// TIA Portal V17 export
// export: Created 2025-07-01T14:25:34.2784289Z, ExportSetting WithDefaults, DisplayName Totally Integrated Automation Portal, DisplayVersion V17 Update 8, DisplayName TIA Portal Openness, DisplayVersion V17 Update 8, DisplayName TIA Portal Version Control Interface, DisplayVersion V17, DisplayName SINAMICS Startdrive Advanced, DisplayVersion V17 SP2, DisplayName SINAMICS Startdrive G110M, G120, G120C, G120D, G120P, G115D, DisplayVersion V17 SP2, DisplayName SINAMICS Startdrive G130, G150, S120, S150, SINAMICS MV, S210, DisplayVersion V17 SP2, DisplayName STEP 7 Professional, DisplayVersion V17 Update 8, DisplayName SINUMERIK ONE STEP 7 Toolbox, DisplayVersion V17 Update 12, DisplayName SINUMERIK ONE PLC Basic Program Plus, DisplayVersion V17 Update 12, DisplayName SINUMERIK 840D sl STEP 7 Toolbox, DisplayVersion V17 Update 12, DisplayName STEP 7 Safety, DisplayVersion V17 Update 6, DisplayName WinCC Advanced, DisplayVersion V17 Update 8
FUNCTION "FC343_NCK_M_CH1_UNIT_1_STA_0" : Void   // FC343, LAD
TITLE = Channel 1 data
{ S7_Optimized_Access := 'FALSE' }
AUTHOR : ETXETAR
VERSION : 1.0
// stored: AutoNumber false, IsIECCheckEnabled false, SetENOAutomatically false, UDAEnableTagReadback false
BEGIN

REGION Network 1: ACKNOWLEDGE M704-UNIT 1 FIXTURE 4 VERIFY PART AND TOOL IS CLAMPED DURING MACHINING (WHEN TRUE DO). TOGGLED / ACKNOWLEDGE M46-VERIFY FIXTURE 1 PART AND TOOL IS CLAMPED DURING
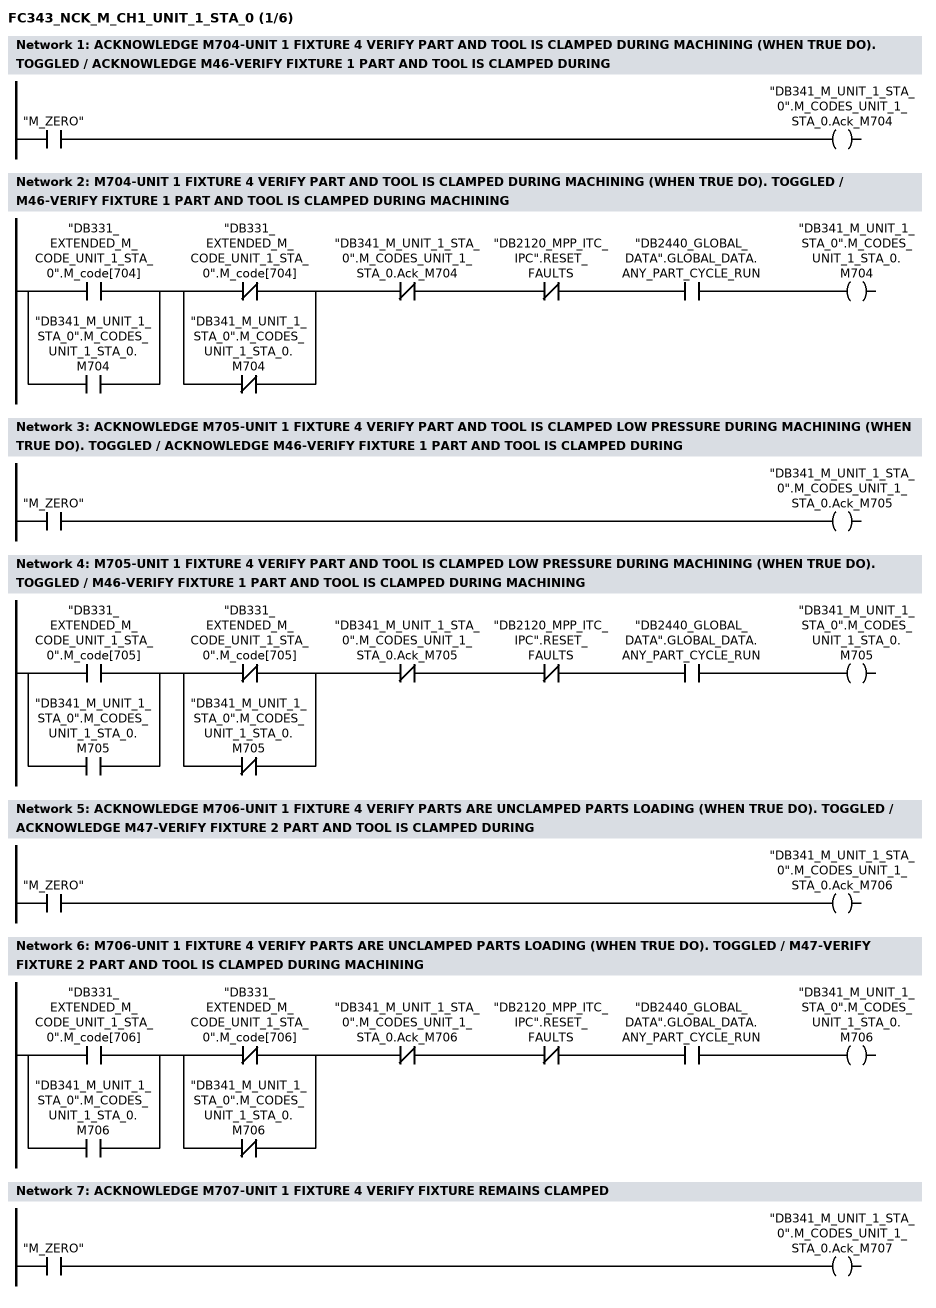
   RUNG wire#powerrail
      Contact( "M_ZERO" )
      Coil( "DB341_M_UNIT_1_STA_0".M_CODES_UNIT_1_STA_0.Ack_M704 )
   END_RUNG
   // the same network as SCL:
   "DB341_M_UNIT_1_STA_0".M_CODES_UNIT_1_STA_0.Ack_M704 := "M_ZERO";
END_REGION

REGION Network 2: M704-UNIT 1 FIXTURE 4 VERIFY PART AND TOOL IS CLAMPED DURING MACHINING (WHEN TRUE DO). TOGGLED / M46-VERIFY FIXTURE 1 PART AND TOOL IS CLAMPED DURING MACHINING
   RUNG wire#powerrail
      Contact( "DB331_EXTENDED_M_CODE_UNIT_1_STA_0".M_code[704] )
      wire#w1
      I_Contact( "DB331_EXTENDED_M_CODE_UNIT_1_STA_0".M_code[704] )
      wire#w2
      I_Contact( "DB341_M_UNIT_1_STA_0".M_CODES_UNIT_1_STA_0.Ack_M704 )
      I_Contact( "DB2120_MPP_ITC_IPC".RESET_FAULTS )
      Contact( "DB2440_GLOBAL_DATA".GLOBAL_DATA.ANY_PART_CYCLE_RUN )
      Coil( "DB341_M_UNIT_1_STA_0".M_CODES_UNIT_1_STA_0.M704 )
   END_RUNG
   RUNG wire#powerrail
      Contact( "DB341_M_UNIT_1_STA_0".M_CODES_UNIT_1_STA_0.M704 )
   END_RUNG wire#w1
   RUNG wire#w1
      I_Contact( "DB341_M_UNIT_1_STA_0".M_CODES_UNIT_1_STA_0.M704 )
   END_RUNG wire#w2
   // the same network as SCL:
   "DB341_M_UNIT_1_STA_0".M_CODES_UNIT_1_STA_0.M704 := ("DB331_EXTENDED_M_CODE_UNIT_1_STA_0".M_code[704] OR "DB341_M_UNIT_1_STA_0".M_CODES_UNIT_1_STA_0.M704) AND (NOT "DB331_EXTENDED_M_CODE_UNIT_1_STA_0".M_code[704] OR NOT "DB341_M_UNIT_1_STA_0".M_CODES_UNIT_1_STA_0.M704) AND NOT "DB341_M_UNIT_1_STA_0".M_CODES_UNIT_1_STA_0.Ack_M704 AND NOT "DB2120_MPP_ITC_IPC".RESET_FAULTS AND "DB2440_GLOBAL_DATA".GLOBAL_DATA.ANY_PART_CYCLE_RUN;
END_REGION

REGION Network 3: ACKNOWLEDGE M705-UNIT 1 FIXTURE 4 VERIFY PART AND TOOL IS CLAMPED LOW PRESSURE DURING MACHINING (WHEN TRUE DO). TOGGLED / ACKNOWLEDGE M46-VERIFY FIXTURE 1 PART AND TOOL IS CLAMPED DURING
   RUNG wire#powerrail
      Contact( "M_ZERO" )
      Coil( "DB341_M_UNIT_1_STA_0".M_CODES_UNIT_1_STA_0.Ack_M705 )
   END_RUNG
   // the same network as SCL:
   "DB341_M_UNIT_1_STA_0".M_CODES_UNIT_1_STA_0.Ack_M705 := "M_ZERO";
END_REGION

REGION Network 4: M705-UNIT 1 FIXTURE 4 VERIFY PART AND TOOL IS CLAMPED LOW PRESSURE DURING MACHINING (WHEN TRUE DO). TOGGLED / M46-VERIFY FIXTURE 1 PART AND TOOL IS CLAMPED DURING MACHINING
   RUNG wire#powerrail
      Contact( "DB331_EXTENDED_M_CODE_UNIT_1_STA_0".M_code[705] )
      wire#w1
      I_Contact( "DB331_EXTENDED_M_CODE_UNIT_1_STA_0".M_code[705] )
      wire#w2
      I_Contact( "DB341_M_UNIT_1_STA_0".M_CODES_UNIT_1_STA_0.Ack_M705 )
      I_Contact( "DB2120_MPP_ITC_IPC".RESET_FAULTS )
      Contact( "DB2440_GLOBAL_DATA".GLOBAL_DATA.ANY_PART_CYCLE_RUN )
      Coil( "DB341_M_UNIT_1_STA_0".M_CODES_UNIT_1_STA_0.M705 )
   END_RUNG
   RUNG wire#powerrail
      Contact( "DB341_M_UNIT_1_STA_0".M_CODES_UNIT_1_STA_0.M705 )
   END_RUNG wire#w1
   RUNG wire#w1
      I_Contact( "DB341_M_UNIT_1_STA_0".M_CODES_UNIT_1_STA_0.M705 )
   END_RUNG wire#w2
   // the same network as SCL:
   "DB341_M_UNIT_1_STA_0".M_CODES_UNIT_1_STA_0.M705 := ("DB331_EXTENDED_M_CODE_UNIT_1_STA_0".M_code[705] OR "DB341_M_UNIT_1_STA_0".M_CODES_UNIT_1_STA_0.M705) AND (NOT "DB331_EXTENDED_M_CODE_UNIT_1_STA_0".M_code[705] OR NOT "DB341_M_UNIT_1_STA_0".M_CODES_UNIT_1_STA_0.M705) AND NOT "DB341_M_UNIT_1_STA_0".M_CODES_UNIT_1_STA_0.Ack_M705 AND NOT "DB2120_MPP_ITC_IPC".RESET_FAULTS AND "DB2440_GLOBAL_DATA".GLOBAL_DATA.ANY_PART_CYCLE_RUN;
END_REGION

REGION Network 5: ACKNOWLEDGE M706-UNIT 1 FIXTURE 4 VERIFY PARTS ARE UNCLAMPED PARTS LOADING (WHEN TRUE DO). TOGGLED / ACKNOWLEDGE M47-VERIFY FIXTURE 2 PART AND TOOL IS CLAMPED DURING
   RUNG wire#powerrail
      Contact( "M_ZERO" )
      Coil( "DB341_M_UNIT_1_STA_0".M_CODES_UNIT_1_STA_0.Ack_M706 )
   END_RUNG
   // the same network as SCL:
   "DB341_M_UNIT_1_STA_0".M_CODES_UNIT_1_STA_0.Ack_M706 := "M_ZERO";
END_REGION

REGION Network 6: M706-UNIT 1 FIXTURE 4 VERIFY PARTS ARE UNCLAMPED PARTS LOADING (WHEN TRUE DO). TOGGLED / M47-VERIFY FIXTURE 2 PART AND TOOL IS CLAMPED DURING MACHINING
   RUNG wire#powerrail
      Contact( "DB331_EXTENDED_M_CODE_UNIT_1_STA_0".M_code[706] )
      wire#w1
      I_Contact( "DB331_EXTENDED_M_CODE_UNIT_1_STA_0".M_code[706] )
      wire#w2
      I_Contact( "DB341_M_UNIT_1_STA_0".M_CODES_UNIT_1_STA_0.Ack_M706 )
      I_Contact( "DB2120_MPP_ITC_IPC".RESET_FAULTS )
      Contact( "DB2440_GLOBAL_DATA".GLOBAL_DATA.ANY_PART_CYCLE_RUN )
      Coil( "DB341_M_UNIT_1_STA_0".M_CODES_UNIT_1_STA_0.M706 )
   END_RUNG
   RUNG wire#powerrail
      Contact( "DB341_M_UNIT_1_STA_0".M_CODES_UNIT_1_STA_0.M706 )
   END_RUNG wire#w1
   RUNG wire#w1
      I_Contact( "DB341_M_UNIT_1_STA_0".M_CODES_UNIT_1_STA_0.M706 )
   END_RUNG wire#w2
   // the same network as SCL:
   "DB341_M_UNIT_1_STA_0".M_CODES_UNIT_1_STA_0.M706 := ("DB331_EXTENDED_M_CODE_UNIT_1_STA_0".M_code[706] OR "DB341_M_UNIT_1_STA_0".M_CODES_UNIT_1_STA_0.M706) AND (NOT "DB331_EXTENDED_M_CODE_UNIT_1_STA_0".M_code[706] OR NOT "DB341_M_UNIT_1_STA_0".M_CODES_UNIT_1_STA_0.M706) AND NOT "DB341_M_UNIT_1_STA_0".M_CODES_UNIT_1_STA_0.Ack_M706 AND NOT "DB2120_MPP_ITC_IPC".RESET_FAULTS AND "DB2440_GLOBAL_DATA".GLOBAL_DATA.ANY_PART_CYCLE_RUN;
END_REGION

REGION Network 7: ACKNOWLEDGE M707-UNIT 1 FIXTURE 4 VERIFY FIXTURE REMAINS CLAMPED
   RUNG wire#powerrail
      Contact( "M_ZERO" )
      Coil( "DB341_M_UNIT_1_STA_0".M_CODES_UNIT_1_STA_0.Ack_M707 )
   END_RUNG
   // the same network as SCL:
   "DB341_M_UNIT_1_STA_0".M_CODES_UNIT_1_STA_0.Ack_M707 := "M_ZERO";
END_REGION

REGION Network 8: M707-UNIT 1 FIXTURE 4 VERIFY FIXTURE REMAINS CLAMPED
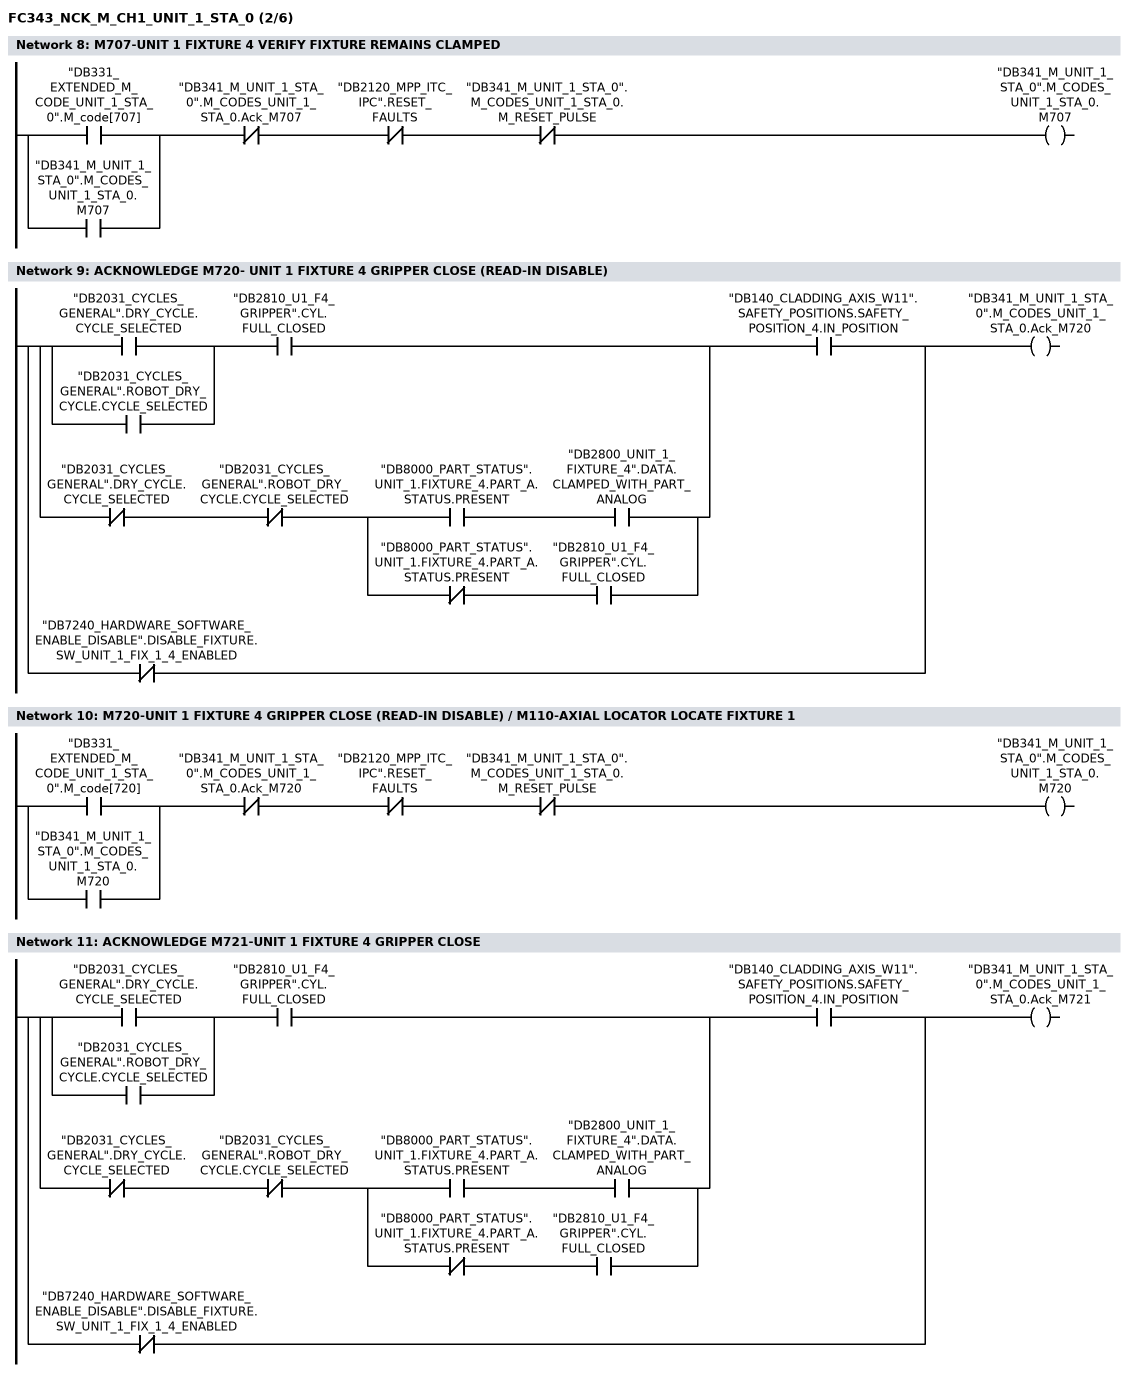
   RUNG wire#powerrail
      Contact( "DB331_EXTENDED_M_CODE_UNIT_1_STA_0".M_code[707] )
      wire#w1
      I_Contact( "DB341_M_UNIT_1_STA_0".M_CODES_UNIT_1_STA_0.Ack_M707 )
      I_Contact( "DB2120_MPP_ITC_IPC".RESET_FAULTS )
      I_Contact( "DB341_M_UNIT_1_STA_0".M_CODES_UNIT_1_STA_0.M_RESET_PULSE )
      Coil( "DB341_M_UNIT_1_STA_0".M_CODES_UNIT_1_STA_0.M707 )
   END_RUNG
   RUNG wire#powerrail
      Contact( "DB341_M_UNIT_1_STA_0".M_CODES_UNIT_1_STA_0.M707 )
   END_RUNG wire#w1
   // the same network as SCL:
   "DB341_M_UNIT_1_STA_0".M_CODES_UNIT_1_STA_0.M707 := ("DB331_EXTENDED_M_CODE_UNIT_1_STA_0".M_code[707] OR "DB341_M_UNIT_1_STA_0".M_CODES_UNIT_1_STA_0.M707) AND NOT "DB341_M_UNIT_1_STA_0".M_CODES_UNIT_1_STA_0.Ack_M707 AND NOT "DB2120_MPP_ITC_IPC".RESET_FAULTS AND NOT "DB341_M_UNIT_1_STA_0".M_CODES_UNIT_1_STA_0.M_RESET_PULSE;
END_REGION

REGION Network 9: ACKNOWLEDGE M720- UNIT 1 FIXTURE 4 GRIPPER CLOSE (READ-IN DISABLE)
   RUNG wire#powerrail
      Contact( "DB2031_CYCLES_GENERAL".DRY_CYCLE.CYCLE_SELECTED )
      wire#w1
      Contact( "DB2810_U1_F4_GRIPPER".CYL.FULL_CLOSED )
      wire#w2
      Contact( "DB140_CLADDING_AXIS_W11".SAFETY_POSITIONS.SAFETY_POSITION_4.IN_POSITION )
      wire#w4
      Coil( "DB341_M_UNIT_1_STA_0".M_CODES_UNIT_1_STA_0.Ack_M720 )
   END_RUNG
   RUNG wire#powerrail
      Contact( "DB2031_CYCLES_GENERAL".ROBOT_DRY_CYCLE.CYCLE_SELECTED )
   END_RUNG wire#w1
   RUNG wire#powerrail
      I_Contact( "DB2031_CYCLES_GENERAL".DRY_CYCLE.CYCLE_SELECTED )
      I_Contact( "DB2031_CYCLES_GENERAL".ROBOT_DRY_CYCLE.CYCLE_SELECTED )
      wire#w3
      Contact( "DB8000_PART_STATUS".UNIT_1.FIXTURE_4.PART_A.STATUS.PRESENT )
      Contact( "DB2800_UNIT_1_FIXTURE_4".DATA.CLAMPED_WITH_PART_ANALOG )
   END_RUNG wire#w2
   RUNG wire#w3
      I_Contact( "DB8000_PART_STATUS".UNIT_1.FIXTURE_4.PART_A.STATUS.PRESENT )
      Contact( "DB2810_U1_F4_GRIPPER".CYL.FULL_CLOSED )
   END_RUNG wire#w2
   RUNG wire#powerrail
      I_Contact( "DB7240_HARDWARE_SOFTWARE_ENABLE_DISABLE".DISABLE_FIXTURE.SW_UNIT_1_FIX_1_4_ENABLED )
   END_RUNG wire#w4
   // the same network as SCL:
   "DB341_M_UNIT_1_STA_0".M_CODES_UNIT_1_STA_0.Ack_M720 := (((("DB2031_CYCLES_GENERAL".DRY_CYCLE.CYCLE_SELECTED OR "DB2031_CYCLES_GENERAL".ROBOT_DRY_CYCLE.CYCLE_SELECTED) AND "DB2810_U1_F4_GRIPPER".CYL.FULL_CLOSED) OR (NOT "DB2031_CYCLES_GENERAL".DRY_CYCLE.CYCLE_SELECTED AND NOT "DB2031_CYCLES_GENERAL".ROBOT_DRY_CYCLE.CYCLE_SELECTED AND (("DB8000_PART_STATUS".UNIT_1.FIXTURE_4.PART_A.STATUS.PRESENT AND "DB2800_UNIT_1_FIXTURE_4".DATA.CLAMPED_WITH_PART_ANALOG) OR (NOT "DB8000_PART_STATUS".UNIT_1.FIXTURE_4.PART_A.STATUS.PRESENT AND "DB2810_U1_F4_GRIPPER".CYL.FULL_CLOSED)))) AND "DB140_CLADDING_AXIS_W11".SAFETY_POSITIONS.SAFETY_POSITION_4.IN_POSITION) OR NOT "DB7240_HARDWARE_SOFTWARE_ENABLE_DISABLE".DISABLE_FIXTURE.SW_UNIT_1_FIX_1_4_ENABLED;
END_REGION

REGION Network 10: M720-UNIT 1 FIXTURE 4 GRIPPER CLOSE (READ-IN DISABLE) / M110-AXIAL LOCATOR LOCATE FIXTURE 1
   RUNG wire#powerrail
      Contact( "DB331_EXTENDED_M_CODE_UNIT_1_STA_0".M_code[720] )
      wire#w1
      I_Contact( "DB341_M_UNIT_1_STA_0".M_CODES_UNIT_1_STA_0.Ack_M720 )
      I_Contact( "DB2120_MPP_ITC_IPC".RESET_FAULTS )
      I_Contact( "DB341_M_UNIT_1_STA_0".M_CODES_UNIT_1_STA_0.M_RESET_PULSE )
      Coil( "DB341_M_UNIT_1_STA_0".M_CODES_UNIT_1_STA_0.M720 )
   END_RUNG
   RUNG wire#powerrail
      Contact( "DB341_M_UNIT_1_STA_0".M_CODES_UNIT_1_STA_0.M720 )
   END_RUNG wire#w1
   // the same network as SCL:
   "DB341_M_UNIT_1_STA_0".M_CODES_UNIT_1_STA_0.M720 := ("DB331_EXTENDED_M_CODE_UNIT_1_STA_0".M_code[720] OR "DB341_M_UNIT_1_STA_0".M_CODES_UNIT_1_STA_0.M720) AND NOT "DB341_M_UNIT_1_STA_0".M_CODES_UNIT_1_STA_0.Ack_M720 AND NOT "DB2120_MPP_ITC_IPC".RESET_FAULTS AND NOT "DB341_M_UNIT_1_STA_0".M_CODES_UNIT_1_STA_0.M_RESET_PULSE;
END_REGION

REGION Network 11: ACKNOWLEDGE M721-UNIT 1 FIXTURE 4 GRIPPER CLOSE
   RUNG wire#powerrail
      Contact( "DB2031_CYCLES_GENERAL".DRY_CYCLE.CYCLE_SELECTED )
      wire#w1
      Contact( "DB2810_U1_F4_GRIPPER".CYL.FULL_CLOSED )
      wire#w2
      Contact( "DB140_CLADDING_AXIS_W11".SAFETY_POSITIONS.SAFETY_POSITION_4.IN_POSITION )
      wire#w4
      Coil( "DB341_M_UNIT_1_STA_0".M_CODES_UNIT_1_STA_0.Ack_M721 )
   END_RUNG
   RUNG wire#powerrail
      Contact( "DB2031_CYCLES_GENERAL".ROBOT_DRY_CYCLE.CYCLE_SELECTED )
   END_RUNG wire#w1
   RUNG wire#powerrail
      I_Contact( "DB2031_CYCLES_GENERAL".DRY_CYCLE.CYCLE_SELECTED )
      I_Contact( "DB2031_CYCLES_GENERAL".ROBOT_DRY_CYCLE.CYCLE_SELECTED )
      wire#w3
      Contact( "DB8000_PART_STATUS".UNIT_1.FIXTURE_4.PART_A.STATUS.PRESENT )
      Contact( "DB2800_UNIT_1_FIXTURE_4".DATA.CLAMPED_WITH_PART_ANALOG )
   END_RUNG wire#w2
   RUNG wire#w3
      I_Contact( "DB8000_PART_STATUS".UNIT_1.FIXTURE_4.PART_A.STATUS.PRESENT )
      Contact( "DB2810_U1_F4_GRIPPER".CYL.FULL_CLOSED )
   END_RUNG wire#w2
   RUNG wire#powerrail
      I_Contact( "DB7240_HARDWARE_SOFTWARE_ENABLE_DISABLE".DISABLE_FIXTURE.SW_UNIT_1_FIX_1_4_ENABLED )
   END_RUNG wire#w4
   // the same network as SCL:
   "DB341_M_UNIT_1_STA_0".M_CODES_UNIT_1_STA_0.Ack_M721 := (((("DB2031_CYCLES_GENERAL".DRY_CYCLE.CYCLE_SELECTED OR "DB2031_CYCLES_GENERAL".ROBOT_DRY_CYCLE.CYCLE_SELECTED) AND "DB2810_U1_F4_GRIPPER".CYL.FULL_CLOSED) OR (NOT "DB2031_CYCLES_GENERAL".DRY_CYCLE.CYCLE_SELECTED AND NOT "DB2031_CYCLES_GENERAL".ROBOT_DRY_CYCLE.CYCLE_SELECTED AND (("DB8000_PART_STATUS".UNIT_1.FIXTURE_4.PART_A.STATUS.PRESENT AND "DB2800_UNIT_1_FIXTURE_4".DATA.CLAMPED_WITH_PART_ANALOG) OR (NOT "DB8000_PART_STATUS".UNIT_1.FIXTURE_4.PART_A.STATUS.PRESENT AND "DB2810_U1_F4_GRIPPER".CYL.FULL_CLOSED)))) AND "DB140_CLADDING_AXIS_W11".SAFETY_POSITIONS.SAFETY_POSITION_4.IN_POSITION) OR NOT "DB7240_HARDWARE_SOFTWARE_ENABLE_DISABLE".DISABLE_FIXTURE.SW_UNIT_1_FIX_1_4_ENABLED;
END_REGION

REGION Network 12: M721-UNIT 1 FIXTURE 4 GRIPPER CLOSE / M110-AXIAL LOCATOR LOCATE FIXTURE 1
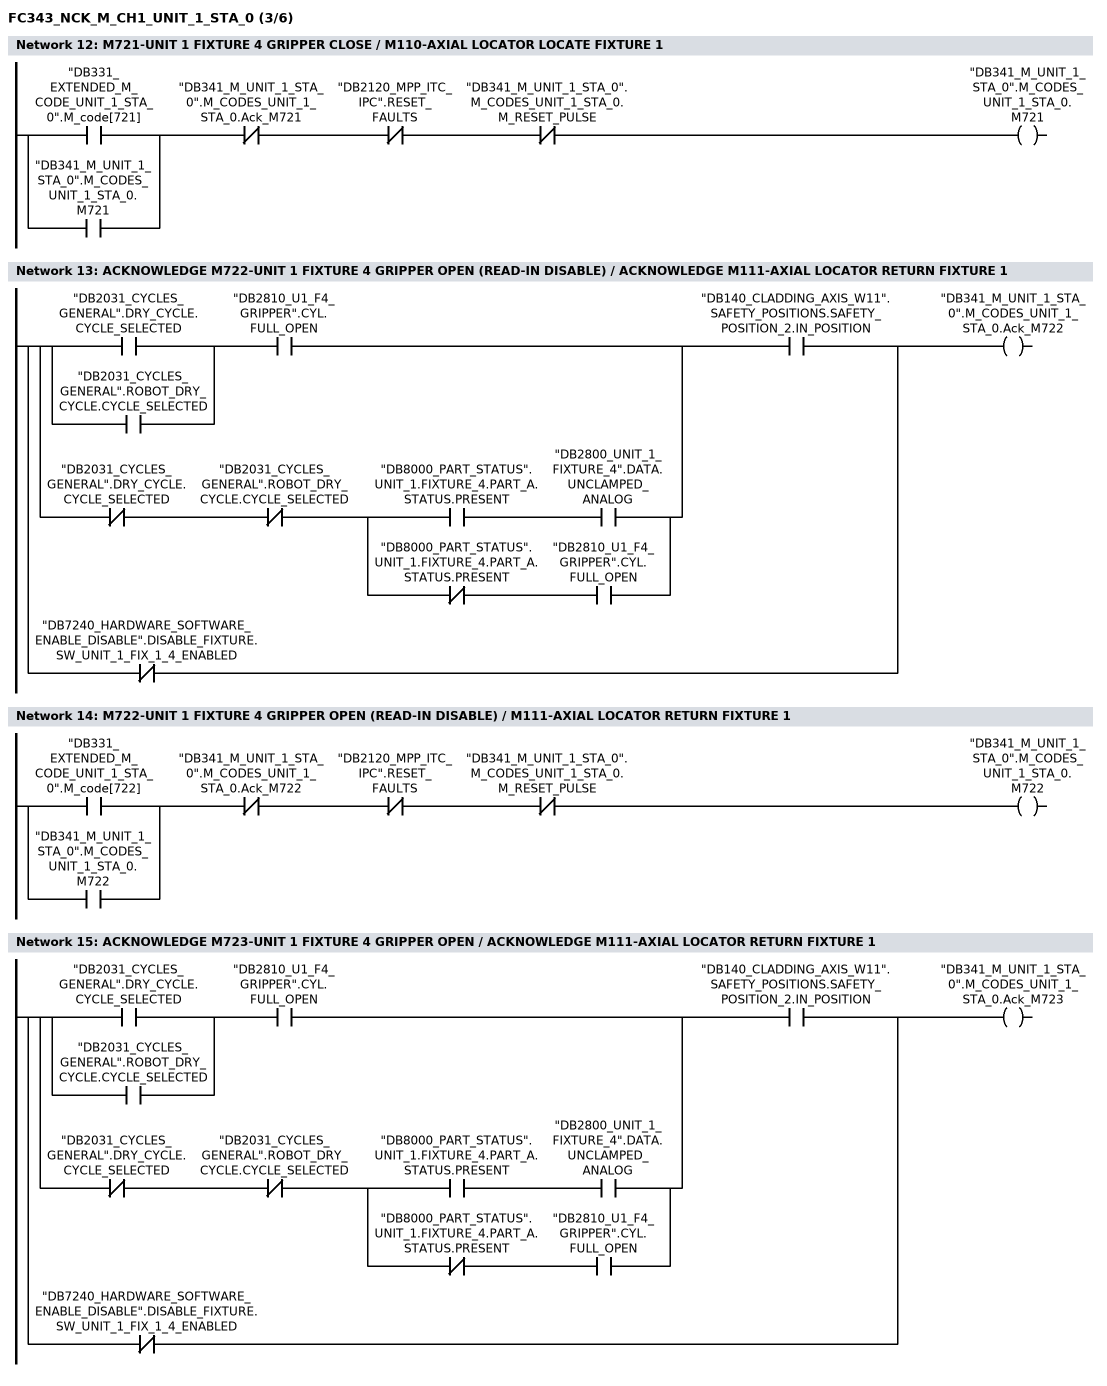
   RUNG wire#powerrail
      Contact( "DB331_EXTENDED_M_CODE_UNIT_1_STA_0".M_code[721] )
      wire#w1
      I_Contact( "DB341_M_UNIT_1_STA_0".M_CODES_UNIT_1_STA_0.Ack_M721 )
      I_Contact( "DB2120_MPP_ITC_IPC".RESET_FAULTS )
      I_Contact( "DB341_M_UNIT_1_STA_0".M_CODES_UNIT_1_STA_0.M_RESET_PULSE )
      Coil( "DB341_M_UNIT_1_STA_0".M_CODES_UNIT_1_STA_0.M721 )
   END_RUNG
   RUNG wire#powerrail
      Contact( "DB341_M_UNIT_1_STA_0".M_CODES_UNIT_1_STA_0.M721 )
   END_RUNG wire#w1
   // the same network as SCL:
   "DB341_M_UNIT_1_STA_0".M_CODES_UNIT_1_STA_0.M721 := ("DB331_EXTENDED_M_CODE_UNIT_1_STA_0".M_code[721] OR "DB341_M_UNIT_1_STA_0".M_CODES_UNIT_1_STA_0.M721) AND NOT "DB341_M_UNIT_1_STA_0".M_CODES_UNIT_1_STA_0.Ack_M721 AND NOT "DB2120_MPP_ITC_IPC".RESET_FAULTS AND NOT "DB341_M_UNIT_1_STA_0".M_CODES_UNIT_1_STA_0.M_RESET_PULSE;
END_REGION

REGION Network 13: ACKNOWLEDGE M722-UNIT 1 FIXTURE 4 GRIPPER OPEN (READ-IN DISABLE) / ACKNOWLEDGE M111-AXIAL LOCATOR RETURN FIXTURE 1
   RUNG wire#powerrail
      Contact( "DB2031_CYCLES_GENERAL".DRY_CYCLE.CYCLE_SELECTED )
      wire#w1
      Contact( "DB2810_U1_F4_GRIPPER".CYL.FULL_OPEN )
      wire#w2
      Contact( "DB140_CLADDING_AXIS_W11".SAFETY_POSITIONS.SAFETY_POSITION_2.IN_POSITION )
      wire#w4
      Coil( "DB341_M_UNIT_1_STA_0".M_CODES_UNIT_1_STA_0.Ack_M722 )
   END_RUNG
   RUNG wire#powerrail
      Contact( "DB2031_CYCLES_GENERAL".ROBOT_DRY_CYCLE.CYCLE_SELECTED )
   END_RUNG wire#w1
   RUNG wire#powerrail
      I_Contact( "DB2031_CYCLES_GENERAL".DRY_CYCLE.CYCLE_SELECTED )
      I_Contact( "DB2031_CYCLES_GENERAL".ROBOT_DRY_CYCLE.CYCLE_SELECTED )
      wire#w3
      Contact( "DB8000_PART_STATUS".UNIT_1.FIXTURE_4.PART_A.STATUS.PRESENT )
      Contact( "DB2800_UNIT_1_FIXTURE_4".DATA.UNCLAMPED_ANALOG )
   END_RUNG wire#w2
   RUNG wire#w3
      I_Contact( "DB8000_PART_STATUS".UNIT_1.FIXTURE_4.PART_A.STATUS.PRESENT )
      Contact( "DB2810_U1_F4_GRIPPER".CYL.FULL_OPEN )
   END_RUNG wire#w2
   RUNG wire#powerrail
      I_Contact( "DB7240_HARDWARE_SOFTWARE_ENABLE_DISABLE".DISABLE_FIXTURE.SW_UNIT_1_FIX_1_4_ENABLED )
   END_RUNG wire#w4
   // the same network as SCL:
   "DB341_M_UNIT_1_STA_0".M_CODES_UNIT_1_STA_0.Ack_M722 := (((("DB2031_CYCLES_GENERAL".DRY_CYCLE.CYCLE_SELECTED OR "DB2031_CYCLES_GENERAL".ROBOT_DRY_CYCLE.CYCLE_SELECTED) AND "DB2810_U1_F4_GRIPPER".CYL.FULL_OPEN) OR (NOT "DB2031_CYCLES_GENERAL".DRY_CYCLE.CYCLE_SELECTED AND NOT "DB2031_CYCLES_GENERAL".ROBOT_DRY_CYCLE.CYCLE_SELECTED AND (("DB8000_PART_STATUS".UNIT_1.FIXTURE_4.PART_A.STATUS.PRESENT AND "DB2800_UNIT_1_FIXTURE_4".DATA.UNCLAMPED_ANALOG) OR (NOT "DB8000_PART_STATUS".UNIT_1.FIXTURE_4.PART_A.STATUS.PRESENT AND "DB2810_U1_F4_GRIPPER".CYL.FULL_OPEN)))) AND "DB140_CLADDING_AXIS_W11".SAFETY_POSITIONS.SAFETY_POSITION_2.IN_POSITION) OR NOT "DB7240_HARDWARE_SOFTWARE_ENABLE_DISABLE".DISABLE_FIXTURE.SW_UNIT_1_FIX_1_4_ENABLED;
END_REGION

REGION Network 14: M722-UNIT 1 FIXTURE 4 GRIPPER OPEN (READ-IN DISABLE) / M111-AXIAL LOCATOR RETURN FIXTURE 1
   RUNG wire#powerrail
      Contact( "DB331_EXTENDED_M_CODE_UNIT_1_STA_0".M_code[722] )
      wire#w1
      I_Contact( "DB341_M_UNIT_1_STA_0".M_CODES_UNIT_1_STA_0.Ack_M722 )
      I_Contact( "DB2120_MPP_ITC_IPC".RESET_FAULTS )
      I_Contact( "DB341_M_UNIT_1_STA_0".M_CODES_UNIT_1_STA_0.M_RESET_PULSE )
      Coil( "DB341_M_UNIT_1_STA_0".M_CODES_UNIT_1_STA_0.M722 )
   END_RUNG
   RUNG wire#powerrail
      Contact( "DB341_M_UNIT_1_STA_0".M_CODES_UNIT_1_STA_0.M722 )
   END_RUNG wire#w1
   // the same network as SCL:
   "DB341_M_UNIT_1_STA_0".M_CODES_UNIT_1_STA_0.M722 := ("DB331_EXTENDED_M_CODE_UNIT_1_STA_0".M_code[722] OR "DB341_M_UNIT_1_STA_0".M_CODES_UNIT_1_STA_0.M722) AND NOT "DB341_M_UNIT_1_STA_0".M_CODES_UNIT_1_STA_0.Ack_M722 AND NOT "DB2120_MPP_ITC_IPC".RESET_FAULTS AND NOT "DB341_M_UNIT_1_STA_0".M_CODES_UNIT_1_STA_0.M_RESET_PULSE;
END_REGION

REGION Network 15: ACKNOWLEDGE M723-UNIT 1 FIXTURE 4 GRIPPER OPEN / ACKNOWLEDGE M111-AXIAL LOCATOR RETURN FIXTURE 1
   RUNG wire#powerrail
      Contact( "DB2031_CYCLES_GENERAL".DRY_CYCLE.CYCLE_SELECTED )
      wire#w1
      Contact( "DB2810_U1_F4_GRIPPER".CYL.FULL_OPEN )
      wire#w2
      Contact( "DB140_CLADDING_AXIS_W11".SAFETY_POSITIONS.SAFETY_POSITION_2.IN_POSITION )
      wire#w4
      Coil( "DB341_M_UNIT_1_STA_0".M_CODES_UNIT_1_STA_0.Ack_M723 )
   END_RUNG
   RUNG wire#powerrail
      Contact( "DB2031_CYCLES_GENERAL".ROBOT_DRY_CYCLE.CYCLE_SELECTED )
   END_RUNG wire#w1
   RUNG wire#powerrail
      I_Contact( "DB2031_CYCLES_GENERAL".DRY_CYCLE.CYCLE_SELECTED )
      I_Contact( "DB2031_CYCLES_GENERAL".ROBOT_DRY_CYCLE.CYCLE_SELECTED )
      wire#w3
      Contact( "DB8000_PART_STATUS".UNIT_1.FIXTURE_4.PART_A.STATUS.PRESENT )
      Contact( "DB2800_UNIT_1_FIXTURE_4".DATA.UNCLAMPED_ANALOG )
   END_RUNG wire#w2
   RUNG wire#w3
      I_Contact( "DB8000_PART_STATUS".UNIT_1.FIXTURE_4.PART_A.STATUS.PRESENT )
      Contact( "DB2810_U1_F4_GRIPPER".CYL.FULL_OPEN )
   END_RUNG wire#w2
   RUNG wire#powerrail
      I_Contact( "DB7240_HARDWARE_SOFTWARE_ENABLE_DISABLE".DISABLE_FIXTURE.SW_UNIT_1_FIX_1_4_ENABLED )
   END_RUNG wire#w4
   // the same network as SCL:
   "DB341_M_UNIT_1_STA_0".M_CODES_UNIT_1_STA_0.Ack_M723 := (((("DB2031_CYCLES_GENERAL".DRY_CYCLE.CYCLE_SELECTED OR "DB2031_CYCLES_GENERAL".ROBOT_DRY_CYCLE.CYCLE_SELECTED) AND "DB2810_U1_F4_GRIPPER".CYL.FULL_OPEN) OR (NOT "DB2031_CYCLES_GENERAL".DRY_CYCLE.CYCLE_SELECTED AND NOT "DB2031_CYCLES_GENERAL".ROBOT_DRY_CYCLE.CYCLE_SELECTED AND (("DB8000_PART_STATUS".UNIT_1.FIXTURE_4.PART_A.STATUS.PRESENT AND "DB2800_UNIT_1_FIXTURE_4".DATA.UNCLAMPED_ANALOG) OR (NOT "DB8000_PART_STATUS".UNIT_1.FIXTURE_4.PART_A.STATUS.PRESENT AND "DB2810_U1_F4_GRIPPER".CYL.FULL_OPEN)))) AND "DB140_CLADDING_AXIS_W11".SAFETY_POSITIONS.SAFETY_POSITION_2.IN_POSITION) OR NOT "DB7240_HARDWARE_SOFTWARE_ENABLE_DISABLE".DISABLE_FIXTURE.SW_UNIT_1_FIX_1_4_ENABLED;
END_REGION

REGION Network 16: M723-UNIT 1 FIXTURE 4 GRIPPER OPEN / M111-AXIAL LOCATOR RETURN FIXTURE 1
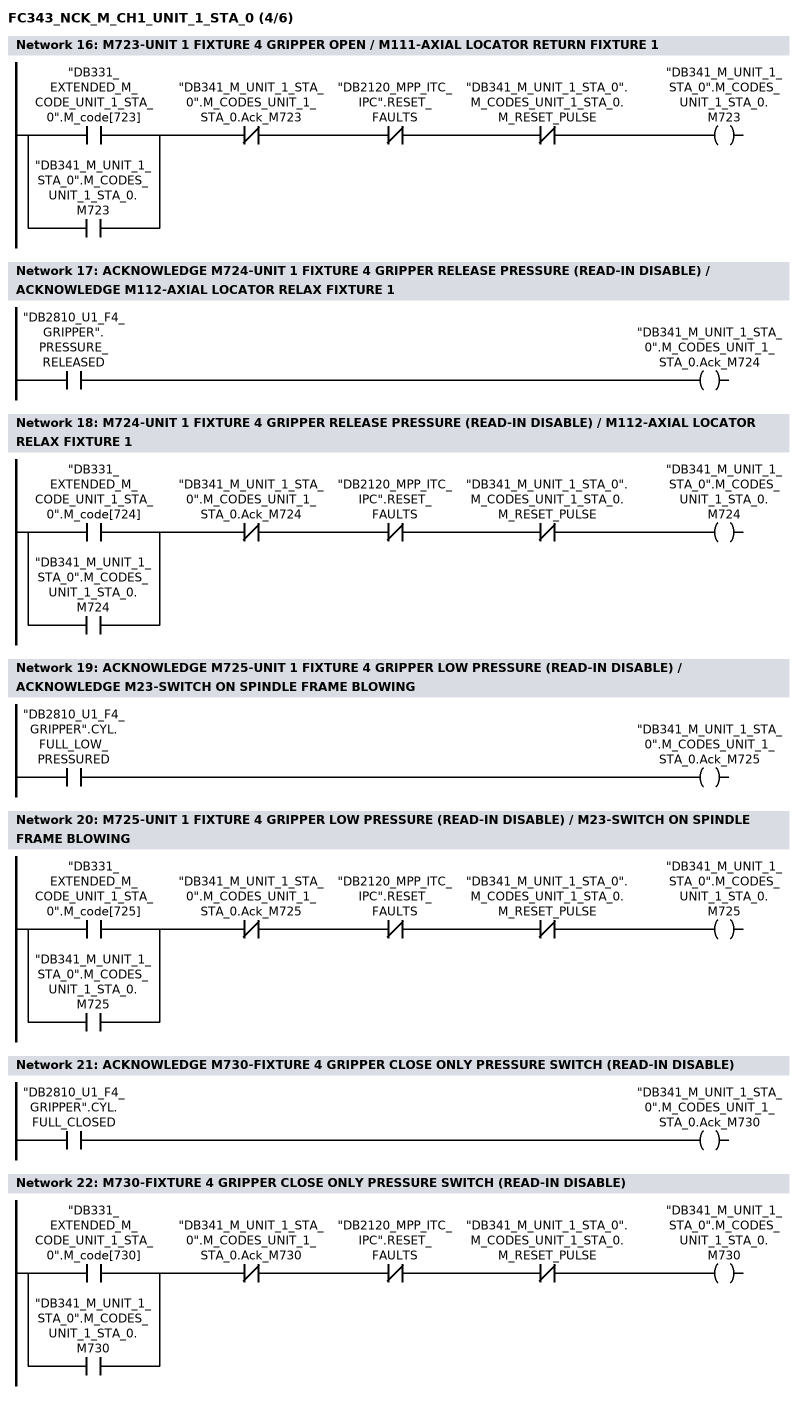
   RUNG wire#powerrail
      Contact( "DB331_EXTENDED_M_CODE_UNIT_1_STA_0".M_code[723] )
      wire#w1
      I_Contact( "DB341_M_UNIT_1_STA_0".M_CODES_UNIT_1_STA_0.Ack_M723 )
      I_Contact( "DB2120_MPP_ITC_IPC".RESET_FAULTS )
      I_Contact( "DB341_M_UNIT_1_STA_0".M_CODES_UNIT_1_STA_0.M_RESET_PULSE )
      Coil( "DB341_M_UNIT_1_STA_0".M_CODES_UNIT_1_STA_0.M723 )
   END_RUNG
   RUNG wire#powerrail
      Contact( "DB341_M_UNIT_1_STA_0".M_CODES_UNIT_1_STA_0.M723 )
   END_RUNG wire#w1
   // the same network as SCL:
   "DB341_M_UNIT_1_STA_0".M_CODES_UNIT_1_STA_0.M723 := ("DB331_EXTENDED_M_CODE_UNIT_1_STA_0".M_code[723] OR "DB341_M_UNIT_1_STA_0".M_CODES_UNIT_1_STA_0.M723) AND NOT "DB341_M_UNIT_1_STA_0".M_CODES_UNIT_1_STA_0.Ack_M723 AND NOT "DB2120_MPP_ITC_IPC".RESET_FAULTS AND NOT "DB341_M_UNIT_1_STA_0".M_CODES_UNIT_1_STA_0.M_RESET_PULSE;
END_REGION

REGION Network 17: ACKNOWLEDGE M724-UNIT 1 FIXTURE 4 GRIPPER RELEASE PRESSURE (READ-IN DISABLE) / ACKNOWLEDGE M112-AXIAL LOCATOR RELAX FIXTURE 1
   RUNG wire#powerrail
      Contact( "DB2810_U1_F4_GRIPPER".PRESSURE_RELEASED )
      Coil( "DB341_M_UNIT_1_STA_0".M_CODES_UNIT_1_STA_0.Ack_M724 )
   END_RUNG
   // the same network as SCL:
   "DB341_M_UNIT_1_STA_0".M_CODES_UNIT_1_STA_0.Ack_M724 := "DB2810_U1_F4_GRIPPER".PRESSURE_RELEASED;
END_REGION

REGION Network 18: M724-UNIT 1 FIXTURE 4 GRIPPER RELEASE PRESSURE (READ-IN DISABLE) / M112-AXIAL LOCATOR RELAX FIXTURE 1
   RUNG wire#powerrail
      Contact( "DB331_EXTENDED_M_CODE_UNIT_1_STA_0".M_code[724] )
      wire#w1
      I_Contact( "DB341_M_UNIT_1_STA_0".M_CODES_UNIT_1_STA_0.Ack_M724 )
      I_Contact( "DB2120_MPP_ITC_IPC".RESET_FAULTS )
      I_Contact( "DB341_M_UNIT_1_STA_0".M_CODES_UNIT_1_STA_0.M_RESET_PULSE )
      Coil( "DB341_M_UNIT_1_STA_0".M_CODES_UNIT_1_STA_0.M724 )
   END_RUNG
   RUNG wire#powerrail
      Contact( "DB341_M_UNIT_1_STA_0".M_CODES_UNIT_1_STA_0.M724 )
   END_RUNG wire#w1
   // the same network as SCL:
   "DB341_M_UNIT_1_STA_0".M_CODES_UNIT_1_STA_0.M724 := ("DB331_EXTENDED_M_CODE_UNIT_1_STA_0".M_code[724] OR "DB341_M_UNIT_1_STA_0".M_CODES_UNIT_1_STA_0.M724) AND NOT "DB341_M_UNIT_1_STA_0".M_CODES_UNIT_1_STA_0.Ack_M724 AND NOT "DB2120_MPP_ITC_IPC".RESET_FAULTS AND NOT "DB341_M_UNIT_1_STA_0".M_CODES_UNIT_1_STA_0.M_RESET_PULSE;
END_REGION

REGION Network 19: ACKNOWLEDGE M725-UNIT 1 FIXTURE 4 GRIPPER LOW PRESSURE (READ-IN DISABLE) / ACKNOWLEDGE M23-SWITCH ON SPINDLE FRAME BLOWING
   RUNG wire#powerrail
      Contact( "DB2810_U1_F4_GRIPPER".CYL.FULL_LOW_PRESSURED )
      Coil( "DB341_M_UNIT_1_STA_0".M_CODES_UNIT_1_STA_0.Ack_M725 )
   END_RUNG
   // the same network as SCL:
   "DB341_M_UNIT_1_STA_0".M_CODES_UNIT_1_STA_0.Ack_M725 := "DB2810_U1_F4_GRIPPER".CYL.FULL_LOW_PRESSURED;
END_REGION

REGION Network 20: M725-UNIT 1 FIXTURE 4 GRIPPER LOW PRESSURE (READ-IN DISABLE) / M23-SWITCH ON SPINDLE FRAME BLOWING
   RUNG wire#powerrail
      Contact( "DB331_EXTENDED_M_CODE_UNIT_1_STA_0".M_code[725] )
      wire#w1
      I_Contact( "DB341_M_UNIT_1_STA_0".M_CODES_UNIT_1_STA_0.Ack_M725 )
      I_Contact( "DB2120_MPP_ITC_IPC".RESET_FAULTS )
      I_Contact( "DB341_M_UNIT_1_STA_0".M_CODES_UNIT_1_STA_0.M_RESET_PULSE )
      Coil( "DB341_M_UNIT_1_STA_0".M_CODES_UNIT_1_STA_0.M725 )
   END_RUNG
   RUNG wire#powerrail
      Contact( "DB341_M_UNIT_1_STA_0".M_CODES_UNIT_1_STA_0.M725 )
   END_RUNG wire#w1
   // the same network as SCL:
   "DB341_M_UNIT_1_STA_0".M_CODES_UNIT_1_STA_0.M725 := ("DB331_EXTENDED_M_CODE_UNIT_1_STA_0".M_code[725] OR "DB341_M_UNIT_1_STA_0".M_CODES_UNIT_1_STA_0.M725) AND NOT "DB341_M_UNIT_1_STA_0".M_CODES_UNIT_1_STA_0.Ack_M725 AND NOT "DB2120_MPP_ITC_IPC".RESET_FAULTS AND NOT "DB341_M_UNIT_1_STA_0".M_CODES_UNIT_1_STA_0.M_RESET_PULSE;
END_REGION

REGION Network 21: ACKNOWLEDGE M730-FIXTURE 4 GRIPPER CLOSE ONLY PRESSURE SWITCH (READ-IN DISABLE)
   RUNG wire#powerrail
      Contact( "DB2810_U1_F4_GRIPPER".CYL.FULL_CLOSED )
      Coil( "DB341_M_UNIT_1_STA_0".M_CODES_UNIT_1_STA_0.Ack_M730 )
   END_RUNG
   // the same network as SCL:
   "DB341_M_UNIT_1_STA_0".M_CODES_UNIT_1_STA_0.Ack_M730 := "DB2810_U1_F4_GRIPPER".CYL.FULL_CLOSED;
END_REGION

REGION Network 22: M730-FIXTURE 4 GRIPPER CLOSE ONLY PRESSURE SWITCH (READ-IN DISABLE)
   RUNG wire#powerrail
      Contact( "DB331_EXTENDED_M_CODE_UNIT_1_STA_0".M_code[730] )
      wire#w1
      I_Contact( "DB341_M_UNIT_1_STA_0".M_CODES_UNIT_1_STA_0.Ack_M730 )
      I_Contact( "DB2120_MPP_ITC_IPC".RESET_FAULTS )
      I_Contact( "DB341_M_UNIT_1_STA_0".M_CODES_UNIT_1_STA_0.M_RESET_PULSE )
      Coil( "DB341_M_UNIT_1_STA_0".M_CODES_UNIT_1_STA_0.M730 )
   END_RUNG
   RUNG wire#powerrail
      Contact( "DB341_M_UNIT_1_STA_0".M_CODES_UNIT_1_STA_0.M730 )
   END_RUNG wire#w1
   // the same network as SCL:
   "DB341_M_UNIT_1_STA_0".M_CODES_UNIT_1_STA_0.M730 := ("DB331_EXTENDED_M_CODE_UNIT_1_STA_0".M_code[730] OR "DB341_M_UNIT_1_STA_0".M_CODES_UNIT_1_STA_0.M730) AND NOT "DB341_M_UNIT_1_STA_0".M_CODES_UNIT_1_STA_0.Ack_M730 AND NOT "DB2120_MPP_ITC_IPC".RESET_FAULTS AND NOT "DB341_M_UNIT_1_STA_0".M_CODES_UNIT_1_STA_0.M_RESET_PULSE;
END_REGION

REGION Network 23: ACKNOWLEDGE M731-FIXTURE 4 GRIPPER CLOSE ONLY PRESSURE SWITCH / ACKNOWLEDGE M23-SWITCH ON SPINDLE FRAME BLOWING
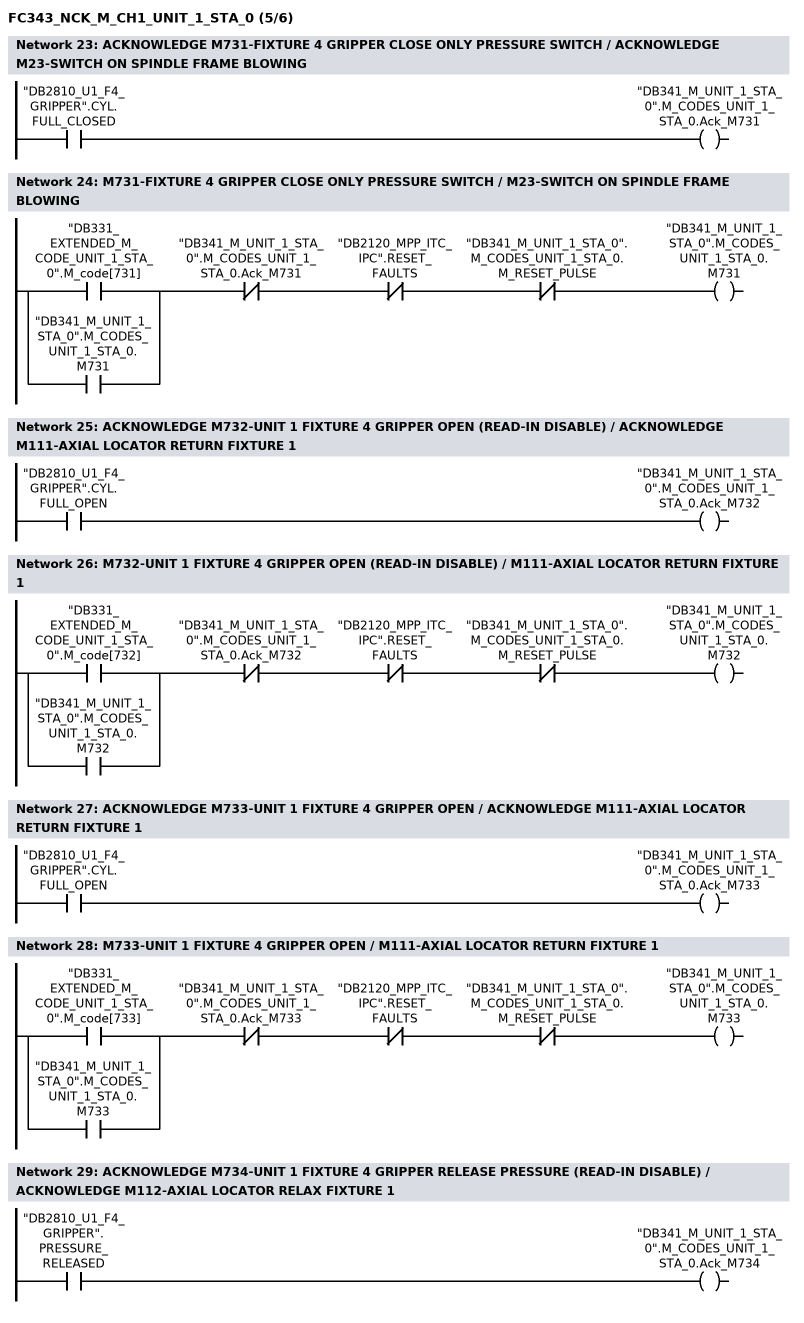
   RUNG wire#powerrail
      Contact( "DB2810_U1_F4_GRIPPER".CYL.FULL_CLOSED )
      Coil( "DB341_M_UNIT_1_STA_0".M_CODES_UNIT_1_STA_0.Ack_M731 )
   END_RUNG
   // the same network as SCL:
   "DB341_M_UNIT_1_STA_0".M_CODES_UNIT_1_STA_0.Ack_M731 := "DB2810_U1_F4_GRIPPER".CYL.FULL_CLOSED;
END_REGION

REGION Network 24: M731-FIXTURE 4 GRIPPER CLOSE ONLY PRESSURE SWITCH / M23-SWITCH ON SPINDLE FRAME BLOWING
   RUNG wire#powerrail
      Contact( "DB331_EXTENDED_M_CODE_UNIT_1_STA_0".M_code[731] )
      wire#w1
      I_Contact( "DB341_M_UNIT_1_STA_0".M_CODES_UNIT_1_STA_0.Ack_M731 )
      I_Contact( "DB2120_MPP_ITC_IPC".RESET_FAULTS )
      I_Contact( "DB341_M_UNIT_1_STA_0".M_CODES_UNIT_1_STA_0.M_RESET_PULSE )
      Coil( "DB341_M_UNIT_1_STA_0".M_CODES_UNIT_1_STA_0.M731 )
   END_RUNG
   RUNG wire#powerrail
      Contact( "DB341_M_UNIT_1_STA_0".M_CODES_UNIT_1_STA_0.M731 )
   END_RUNG wire#w1
   // the same network as SCL:
   "DB341_M_UNIT_1_STA_0".M_CODES_UNIT_1_STA_0.M731 := ("DB331_EXTENDED_M_CODE_UNIT_1_STA_0".M_code[731] OR "DB341_M_UNIT_1_STA_0".M_CODES_UNIT_1_STA_0.M731) AND NOT "DB341_M_UNIT_1_STA_0".M_CODES_UNIT_1_STA_0.Ack_M731 AND NOT "DB2120_MPP_ITC_IPC".RESET_FAULTS AND NOT "DB341_M_UNIT_1_STA_0".M_CODES_UNIT_1_STA_0.M_RESET_PULSE;
END_REGION

REGION Network 25: ACKNOWLEDGE M732-UNIT 1 FIXTURE 4 GRIPPER OPEN (READ-IN DISABLE) / ACKNOWLEDGE M111-AXIAL LOCATOR RETURN FIXTURE 1
   RUNG wire#powerrail
      Contact( "DB2810_U1_F4_GRIPPER".CYL.FULL_OPEN )
      Coil( "DB341_M_UNIT_1_STA_0".M_CODES_UNIT_1_STA_0.Ack_M732 )
   END_RUNG
   // the same network as SCL:
   "DB341_M_UNIT_1_STA_0".M_CODES_UNIT_1_STA_0.Ack_M732 := "DB2810_U1_F4_GRIPPER".CYL.FULL_OPEN;
END_REGION

REGION Network 26: M732-UNIT 1 FIXTURE 4 GRIPPER OPEN (READ-IN DISABLE) / M111-AXIAL LOCATOR RETURN FIXTURE 1
   RUNG wire#powerrail
      Contact( "DB331_EXTENDED_M_CODE_UNIT_1_STA_0".M_code[732] )
      wire#w1
      I_Contact( "DB341_M_UNIT_1_STA_0".M_CODES_UNIT_1_STA_0.Ack_M732 )
      I_Contact( "DB2120_MPP_ITC_IPC".RESET_FAULTS )
      I_Contact( "DB341_M_UNIT_1_STA_0".M_CODES_UNIT_1_STA_0.M_RESET_PULSE )
      Coil( "DB341_M_UNIT_1_STA_0".M_CODES_UNIT_1_STA_0.M732 )
   END_RUNG
   RUNG wire#powerrail
      Contact( "DB341_M_UNIT_1_STA_0".M_CODES_UNIT_1_STA_0.M732 )
   END_RUNG wire#w1
   // the same network as SCL:
   "DB341_M_UNIT_1_STA_0".M_CODES_UNIT_1_STA_0.M732 := ("DB331_EXTENDED_M_CODE_UNIT_1_STA_0".M_code[732] OR "DB341_M_UNIT_1_STA_0".M_CODES_UNIT_1_STA_0.M732) AND NOT "DB341_M_UNIT_1_STA_0".M_CODES_UNIT_1_STA_0.Ack_M732 AND NOT "DB2120_MPP_ITC_IPC".RESET_FAULTS AND NOT "DB341_M_UNIT_1_STA_0".M_CODES_UNIT_1_STA_0.M_RESET_PULSE;
END_REGION

REGION Network 27: ACKNOWLEDGE M733-UNIT 1 FIXTURE 4 GRIPPER OPEN / ACKNOWLEDGE M111-AXIAL LOCATOR RETURN FIXTURE 1
   RUNG wire#powerrail
      Contact( "DB2810_U1_F4_GRIPPER".CYL.FULL_OPEN )
      Coil( "DB341_M_UNIT_1_STA_0".M_CODES_UNIT_1_STA_0.Ack_M733 )
   END_RUNG
   // the same network as SCL:
   "DB341_M_UNIT_1_STA_0".M_CODES_UNIT_1_STA_0.Ack_M733 := "DB2810_U1_F4_GRIPPER".CYL.FULL_OPEN;
END_REGION

REGION Network 28: M733-UNIT 1 FIXTURE 4 GRIPPER OPEN / M111-AXIAL LOCATOR RETURN FIXTURE 1
   RUNG wire#powerrail
      Contact( "DB331_EXTENDED_M_CODE_UNIT_1_STA_0".M_code[733] )
      wire#w1
      I_Contact( "DB341_M_UNIT_1_STA_0".M_CODES_UNIT_1_STA_0.Ack_M733 )
      I_Contact( "DB2120_MPP_ITC_IPC".RESET_FAULTS )
      I_Contact( "DB341_M_UNIT_1_STA_0".M_CODES_UNIT_1_STA_0.M_RESET_PULSE )
      Coil( "DB341_M_UNIT_1_STA_0".M_CODES_UNIT_1_STA_0.M733 )
   END_RUNG
   RUNG wire#powerrail
      Contact( "DB341_M_UNIT_1_STA_0".M_CODES_UNIT_1_STA_0.M733 )
   END_RUNG wire#w1
   // the same network as SCL:
   "DB341_M_UNIT_1_STA_0".M_CODES_UNIT_1_STA_0.M733 := ("DB331_EXTENDED_M_CODE_UNIT_1_STA_0".M_code[733] OR "DB341_M_UNIT_1_STA_0".M_CODES_UNIT_1_STA_0.M733) AND NOT "DB341_M_UNIT_1_STA_0".M_CODES_UNIT_1_STA_0.Ack_M733 AND NOT "DB2120_MPP_ITC_IPC".RESET_FAULTS AND NOT "DB341_M_UNIT_1_STA_0".M_CODES_UNIT_1_STA_0.M_RESET_PULSE;
END_REGION

REGION Network 29: ACKNOWLEDGE M734-UNIT 1 FIXTURE 4 GRIPPER RELEASE PRESSURE (READ-IN DISABLE) / ACKNOWLEDGE M112-AXIAL LOCATOR RELAX FIXTURE 1
   RUNG wire#powerrail
      Contact( "DB2810_U1_F4_GRIPPER".PRESSURE_RELEASED )
      Coil( "DB341_M_UNIT_1_STA_0".M_CODES_UNIT_1_STA_0.Ack_M734 )
   END_RUNG
   // the same network as SCL:
   "DB341_M_UNIT_1_STA_0".M_CODES_UNIT_1_STA_0.Ack_M734 := "DB2810_U1_F4_GRIPPER".PRESSURE_RELEASED;
END_REGION

REGION Network 30: M734-UNIT 1 FIXTURE 4 GRIPPER RELEASE PRESSURE (READ-IN DISABLE) / M112-AXIAL LOCATOR RELAX FIXTURE 1
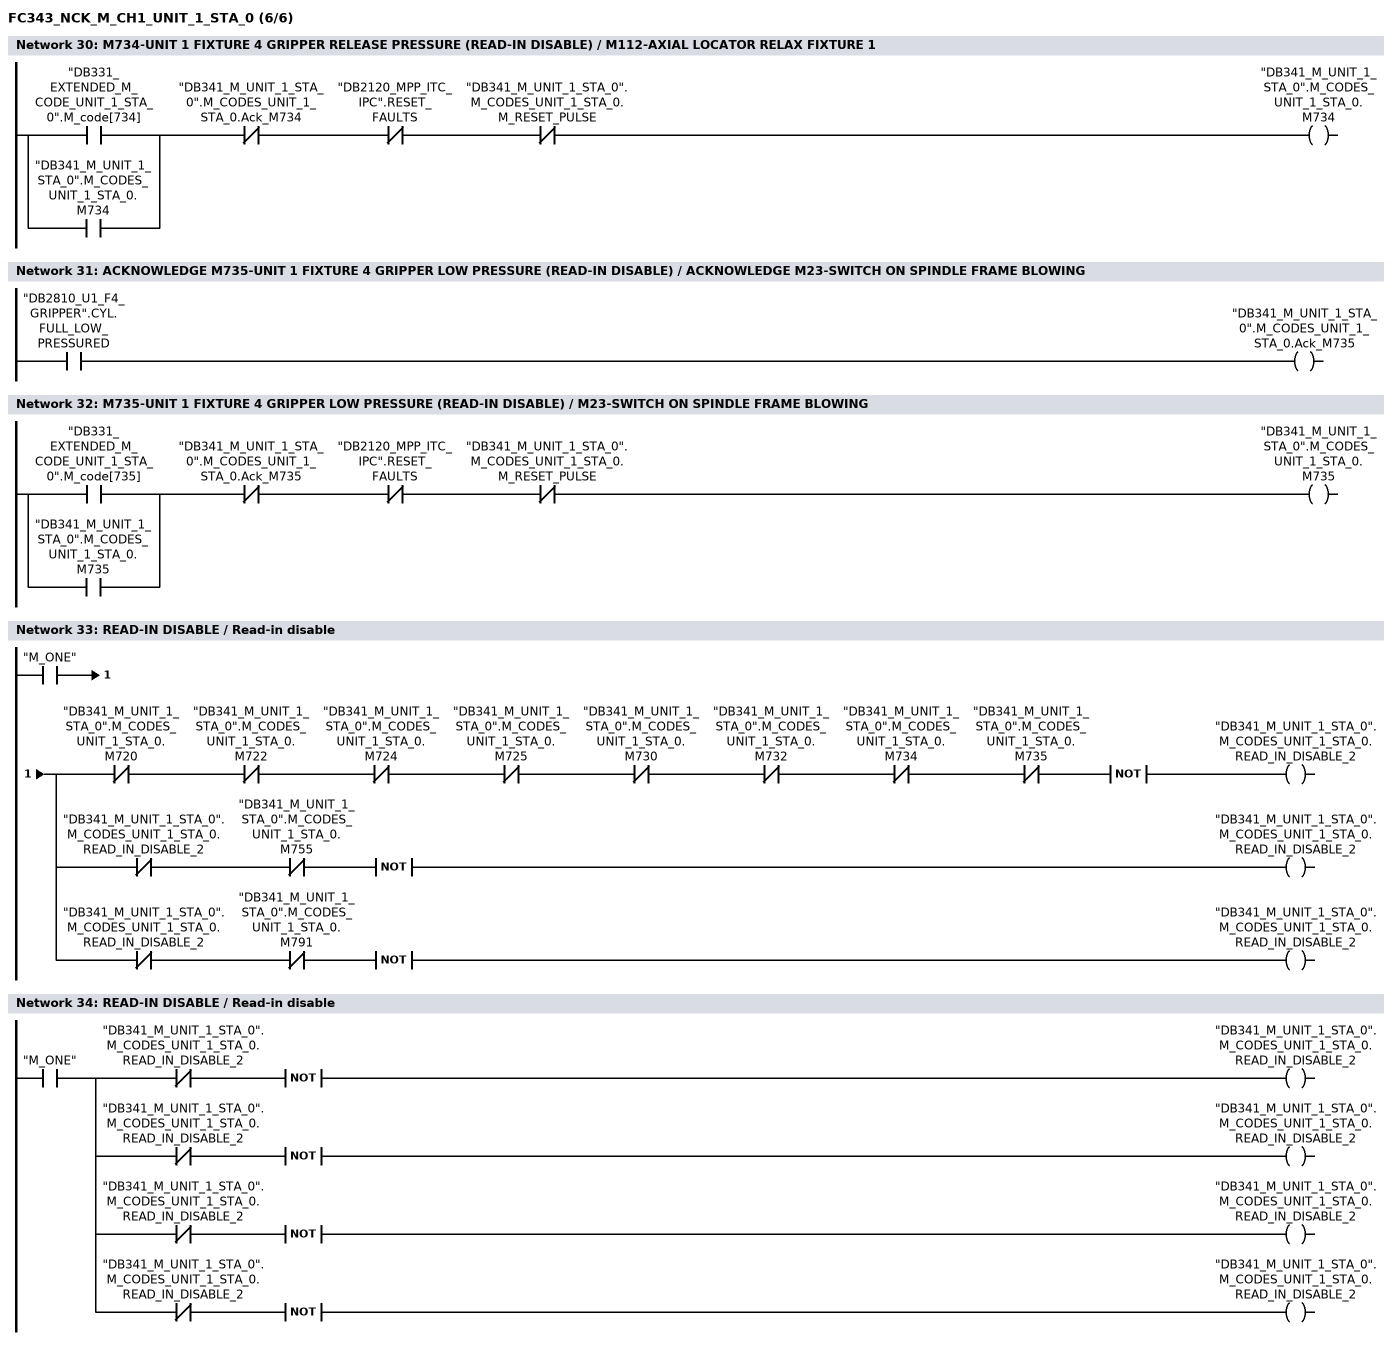
   RUNG wire#powerrail
      Contact( "DB331_EXTENDED_M_CODE_UNIT_1_STA_0".M_code[734] )
      wire#w1
      I_Contact( "DB341_M_UNIT_1_STA_0".M_CODES_UNIT_1_STA_0.Ack_M734 )
      I_Contact( "DB2120_MPP_ITC_IPC".RESET_FAULTS )
      I_Contact( "DB341_M_UNIT_1_STA_0".M_CODES_UNIT_1_STA_0.M_RESET_PULSE )
      Coil( "DB341_M_UNIT_1_STA_0".M_CODES_UNIT_1_STA_0.M734 )
   END_RUNG
   RUNG wire#powerrail
      Contact( "DB341_M_UNIT_1_STA_0".M_CODES_UNIT_1_STA_0.M734 )
   END_RUNG wire#w1
   // the same network as SCL:
   "DB341_M_UNIT_1_STA_0".M_CODES_UNIT_1_STA_0.M734 := ("DB331_EXTENDED_M_CODE_UNIT_1_STA_0".M_code[734] OR "DB341_M_UNIT_1_STA_0".M_CODES_UNIT_1_STA_0.M734) AND NOT "DB341_M_UNIT_1_STA_0".M_CODES_UNIT_1_STA_0.Ack_M734 AND NOT "DB2120_MPP_ITC_IPC".RESET_FAULTS AND NOT "DB341_M_UNIT_1_STA_0".M_CODES_UNIT_1_STA_0.M_RESET_PULSE;
END_REGION

REGION Network 31: ACKNOWLEDGE M735-UNIT 1 FIXTURE 4 GRIPPER LOW PRESSURE (READ-IN DISABLE) / ACKNOWLEDGE M23-SWITCH ON SPINDLE FRAME BLOWING
   RUNG wire#powerrail
      Contact( "DB2810_U1_F4_GRIPPER".CYL.FULL_LOW_PRESSURED )
      Coil( "DB341_M_UNIT_1_STA_0".M_CODES_UNIT_1_STA_0.Ack_M735 )
   END_RUNG
   // the same network as SCL:
   "DB341_M_UNIT_1_STA_0".M_CODES_UNIT_1_STA_0.Ack_M735 := "DB2810_U1_F4_GRIPPER".CYL.FULL_LOW_PRESSURED;
END_REGION

REGION Network 32: M735-UNIT 1 FIXTURE 4 GRIPPER LOW PRESSURE (READ-IN DISABLE) / M23-SWITCH ON SPINDLE FRAME BLOWING
   RUNG wire#powerrail
      Contact( "DB331_EXTENDED_M_CODE_UNIT_1_STA_0".M_code[735] )
      wire#w1
      I_Contact( "DB341_M_UNIT_1_STA_0".M_CODES_UNIT_1_STA_0.Ack_M735 )
      I_Contact( "DB2120_MPP_ITC_IPC".RESET_FAULTS )
      I_Contact( "DB341_M_UNIT_1_STA_0".M_CODES_UNIT_1_STA_0.M_RESET_PULSE )
      Coil( "DB341_M_UNIT_1_STA_0".M_CODES_UNIT_1_STA_0.M735 )
   END_RUNG
   RUNG wire#powerrail
      Contact( "DB341_M_UNIT_1_STA_0".M_CODES_UNIT_1_STA_0.M735 )
   END_RUNG wire#w1
   // the same network as SCL:
   "DB341_M_UNIT_1_STA_0".M_CODES_UNIT_1_STA_0.M735 := ("DB331_EXTENDED_M_CODE_UNIT_1_STA_0".M_code[735] OR "DB341_M_UNIT_1_STA_0".M_CODES_UNIT_1_STA_0.M735) AND NOT "DB341_M_UNIT_1_STA_0".M_CODES_UNIT_1_STA_0.Ack_M735 AND NOT "DB2120_MPP_ITC_IPC".RESET_FAULTS AND NOT "DB341_M_UNIT_1_STA_0".M_CODES_UNIT_1_STA_0.M_RESET_PULSE;
END_REGION

REGION Network 33: READ-IN DISABLE / Read-in disable
   RUNG wire#powerrail
      Contact( "M_ONE" )
      wire#w1
      I_Contact( "DB341_M_UNIT_1_STA_0".M_CODES_UNIT_1_STA_0.M720 )
      I_Contact( "DB341_M_UNIT_1_STA_0".M_CODES_UNIT_1_STA_0.M722 )
      I_Contact( "DB341_M_UNIT_1_STA_0".M_CODES_UNIT_1_STA_0.M724 )
      I_Contact( "DB341_M_UNIT_1_STA_0".M_CODES_UNIT_1_STA_0.M725 )
      I_Contact( "DB341_M_UNIT_1_STA_0".M_CODES_UNIT_1_STA_0.M730 )
      I_Contact( "DB341_M_UNIT_1_STA_0".M_CODES_UNIT_1_STA_0.M732 )
      I_Contact( "DB341_M_UNIT_1_STA_0".M_CODES_UNIT_1_STA_0.M734 )
      I_Contact( "DB341_M_UNIT_1_STA_0".M_CODES_UNIT_1_STA_0.M735 )
      Not()
      Coil( "DB341_M_UNIT_1_STA_0".M_CODES_UNIT_1_STA_0.READ_IN_DISABLE_2 )
   END_RUNG
   RUNG wire#w1
      I_Contact( "DB341_M_UNIT_1_STA_0".M_CODES_UNIT_1_STA_0.READ_IN_DISABLE_2 )
      I_Contact( "DB341_M_UNIT_1_STA_0".M_CODES_UNIT_1_STA_0.M755 )
      Not()
      Coil( "DB341_M_UNIT_1_STA_0".M_CODES_UNIT_1_STA_0.READ_IN_DISABLE_2 )
   END_RUNG
   RUNG wire#w1
      I_Contact( "DB341_M_UNIT_1_STA_0".M_CODES_UNIT_1_STA_0.READ_IN_DISABLE_2 )
      I_Contact( "DB341_M_UNIT_1_STA_0".M_CODES_UNIT_1_STA_0.M791 )
      Not()
      Coil( "DB341_M_UNIT_1_STA_0".M_CODES_UNIT_1_STA_0.READ_IN_DISABLE_2 )
   END_RUNG
   // the same network as SCL:
   "DB341_M_UNIT_1_STA_0".M_CODES_UNIT_1_STA_0.READ_IN_DISABLE_2 := NOT ("M_ONE" AND NOT "DB341_M_UNIT_1_STA_0".M_CODES_UNIT_1_STA_0.M720 AND NOT "DB341_M_UNIT_1_STA_0".M_CODES_UNIT_1_STA_0.M722 AND NOT "DB341_M_UNIT_1_STA_0".M_CODES_UNIT_1_STA_0.M724 AND NOT "DB341_M_UNIT_1_STA_0".M_CODES_UNIT_1_STA_0.M725 AND NOT "DB341_M_UNIT_1_STA_0".M_CODES_UNIT_1_STA_0.M730 AND NOT "DB341_M_UNIT_1_STA_0".M_CODES_UNIT_1_STA_0.M732 AND NOT "DB341_M_UNIT_1_STA_0".M_CODES_UNIT_1_STA_0.M734 AND NOT "DB341_M_UNIT_1_STA_0".M_CODES_UNIT_1_STA_0.M735);
   "DB341_M_UNIT_1_STA_0".M_CODES_UNIT_1_STA_0.READ_IN_DISABLE_2 := NOT ("M_ONE" AND NOT "DB341_M_UNIT_1_STA_0".M_CODES_UNIT_1_STA_0.READ_IN_DISABLE_2 AND NOT "DB341_M_UNIT_1_STA_0".M_CODES_UNIT_1_STA_0.M755);
   "DB341_M_UNIT_1_STA_0".M_CODES_UNIT_1_STA_0.READ_IN_DISABLE_2 := NOT ("M_ONE" AND NOT "DB341_M_UNIT_1_STA_0".M_CODES_UNIT_1_STA_0.READ_IN_DISABLE_2 AND NOT "DB341_M_UNIT_1_STA_0".M_CODES_UNIT_1_STA_0.M791);
END_REGION

REGION Network 34: READ-IN DISABLE / Read-in disable
   RUNG wire#powerrail
      Contact( "M_ONE" )
      wire#w1
      I_Contact( "DB341_M_UNIT_1_STA_0".M_CODES_UNIT_1_STA_0.READ_IN_DISABLE_2 )
      Not()
      Coil( "DB341_M_UNIT_1_STA_0".M_CODES_UNIT_1_STA_0.READ_IN_DISABLE_2 )
   END_RUNG
   RUNG wire#w1
      I_Contact( "DB341_M_UNIT_1_STA_0".M_CODES_UNIT_1_STA_0.READ_IN_DISABLE_2 )
      Not()
      Coil( "DB341_M_UNIT_1_STA_0".M_CODES_UNIT_1_STA_0.READ_IN_DISABLE_2 )
   END_RUNG
   RUNG wire#w1
      I_Contact( "DB341_M_UNIT_1_STA_0".M_CODES_UNIT_1_STA_0.READ_IN_DISABLE_2 )
      Not()
      Coil( "DB341_M_UNIT_1_STA_0".M_CODES_UNIT_1_STA_0.READ_IN_DISABLE_2 )
   END_RUNG
   RUNG wire#w1
      I_Contact( "DB341_M_UNIT_1_STA_0".M_CODES_UNIT_1_STA_0.READ_IN_DISABLE_2 )
      Not()
      Coil( "DB341_M_UNIT_1_STA_0".M_CODES_UNIT_1_STA_0.READ_IN_DISABLE_2 )
   END_RUNG
   // the same network as SCL:
   "DB341_M_UNIT_1_STA_0".M_CODES_UNIT_1_STA_0.READ_IN_DISABLE_2 := NOT ("M_ONE" AND NOT "DB341_M_UNIT_1_STA_0".M_CODES_UNIT_1_STA_0.READ_IN_DISABLE_2);
   "DB341_M_UNIT_1_STA_0".M_CODES_UNIT_1_STA_0.READ_IN_DISABLE_2 := NOT ("M_ONE" AND NOT "DB341_M_UNIT_1_STA_0".M_CODES_UNIT_1_STA_0.READ_IN_DISABLE_2);
   "DB341_M_UNIT_1_STA_0".M_CODES_UNIT_1_STA_0.READ_IN_DISABLE_2 := NOT ("M_ONE" AND NOT "DB341_M_UNIT_1_STA_0".M_CODES_UNIT_1_STA_0.READ_IN_DISABLE_2);
   "DB341_M_UNIT_1_STA_0".M_CODES_UNIT_1_STA_0.READ_IN_DISABLE_2 := NOT ("M_ONE" AND NOT "DB341_M_UNIT_1_STA_0".M_CODES_UNIT_1_STA_0.READ_IN_DISABLE_2);
END_REGION
END_FUNCTION
